FUNCTION F_PosWithinDelta : BOOL
VAR_INPUT
    fPosition: LREAL;
    stPositionState: ST_PositionState;
END_VAR


F_PosWithinDelta := F_PosOverLowerBound(fPosition, stPositionState) AND
                    F_PosUnderUpperBound(fPosition, stPositionState);

END_FUNCTION

(* stored: Version 1.1.0.1
   POU F_PosWithinDelta: Id {5e4b12d9-d7b3-420d-a0c0-3caa211d85b5}, SpecialFunc None *)
